FUNCTION_BLOCK ProductOrder_HMI
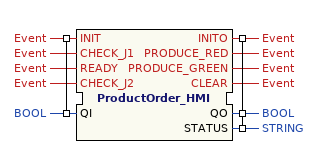
  EVENT_INPUT
    INIT WITH QI;
    CHECK_J1;
    READY;
    CHECK_J2;
  END_EVENT
  EVENT_OUTPUT
    INITO WITH QO, STATUS;
    PRODUCE_RED;
    PRODUCE_GREEN;
    CLEAR;
  END_EVENT
  VAR_INPUT
    QI : BOOL;
  END_VAR
  VAR_OUTPUT
    QO : BOOL;
    STATUS : STRING;
  END_VAR
END_FUNCTION_BLOCK
